Yaskawa INFORM job: R2_W27-A4(90,180)_MP_OK.JBI

/JOB
//NAME R2_W27-A4(90,180)_MP_OK
///FOLDERNAME MP_TEST
//POS
///NPOS 81,81,0,3,0,0
///TOOL 0
///POSTYPE PULSE
///PULSE
C00000=44200,21638,-8218,30156,108783,8626
C00001=67595,-7097,-4564,35957,72928,-14479
C00002=80598,-11631,1969,12944,68774,-20478
C00003=80599,-10712,4409,13031,67770,-20590
C00004=80598,-10715,4407,13031,67770,-20590
C00005=80598,-10719,4404,13032,67770,-20590
C00006=80598,-10715,4407,13031,67770,-20590
C00007=80591,-10742,4386,13033,67770,-20593
C00008=80591,-10741,4387,13033,67770,-20593
C00009=80591,-10742,4386,13033,67770,-20593
C00010=80616,-10653,4455,1959,54638,1214
C00011=74713,-5814,6866,11718,60472,-1274
C00012=77733,-8416,5583,7275,56956,-133
C00013=74892,-4761,7835,12151,60366,-1228
C00014=80616,-10653,4455,1959,54638,1214
C00015=80621,-10639,4466,1958,54638,1216
C00016=80622,-10633,4471,1957,54639,1217
C00017=80626,-10617,4483,1955,54639,1218
C00018=80604,-16221,-12250,12512,75016,-19809
C00019=80613,-16483,-13492,4814,52988,-77020
C00020=80617,-10651,4457,5429,44969,-77444
C00021=80614,-10662,4448,5430,44969,-77445
C00022=79334,-14584,3986,9291,39946,-78705
C00023=81168,-10487,5664,5147,44277,-77224
C00024=80549,-11563,2448,5400,45738,-77430
C00025=81469,-7152,9286,7523,40651,-76865
C00026=81214,-8593,7267,7629,41172,-76947
C00027=79900,-12351,2214,8365,42469,-77481
C00028=78759,-13697,-9805,5892,52278,-77840
C00029=77858,-26804,-24776,6192,54811,-78068
C00030=77858,-26804,-24776,6192,54811,8206
C00031=80560,-10852,4301,23089,88681,-39643
C00032=80562,-10848,4304,23089,88680,-39643
C00033=80600,-11026,3471,23097,89058,-39557
C00034=80047,-12757,2574,23029,88900,-39787
C00035=79798,-9411,5485,22999,88903,-39877
C00036=73696,-20114,6682,31978,77502,-45766
C00037=72021,-21514,1829,31651,80058,-45695
C00038=88031,-24585,-19769,24865,79157,-46389
C00039=74088,-80099,-54440,46439,68409,-50026
C00040=71054,-82284,-78741,37326,78086,-53143
C00041=71054,-82284,-78741,37326,78086,-53143
C00042=141655,19461,21674,-54626,60929,-83209
C00043=140768,21158,24027,-54713,60067,-83168
C00044=140773,21783,25908,-55104,59574,-82809
C00045=140768,21158,24027,-54713,60067,-83168
C00046=156074,19906,-10403,-52836,81444,-87755
C00047=155321,18966,-11276,-52620,81066,-87928
C00048=156074,19906,-10403,-52836,81444,-87755
C00049=158287,-4573,8654,-106143,62454,-35624
C00050=145346,15241,-15914,-44032,85995,9611
C00051=145082,17275,-14042,-43967,85792,9582
C00052=145346,15241,-15914,-44032,85995,9611
C00053=128597,-2596,-22816,-39758,74552,6944
C00054=106236,1119,-8655,-33108,59628,2381
C00055=100502,1007,-8349,-30553,57262,531
C00056=121335,-11193,4016,-73235,33107,-65970
C00057=121314,-11175,4070,-52209,41640,-77705
C00058=121322,-11192,4065,-52217,41640,-77699
C00059=121326,-11199,4064,-52221,41641,-77697
C00060=121319,-11903,2209,-51536,42130,-78112
C00061=122361,-11180,4070,-52628,42228,-77380
C00062=121327,-11199,4064,-52222,41641,-77696
C00063=121327,-11199,4064,-52222,41641,-77696
C00064=121328,-11199,4065,-52223,41641,-77696
C00065=121325,-11192,4067,-52219,41641,-77698
C00066=121317,-11174,4072,-52211,41640,-77704
C00067=121324,-11180,4031,-66023,34984,-69858
C00068=121305,-11164,4064,-33775,34107,58027
C00069=121211,-10931,3851,-41868,44478,53115
C00070=117301,-6994,3549,-31202,46743,49457
C00071=117109,-6013,5862,-33344,45913,49803
C00072=121892,-11860,2463,-42413,44821,53021
C00073=122357,-11331,3957,-43061,44562,53464
C00074=117366,750,11411,-33444,46067,49884
C00075=119475,-2324,8124,-34252,47278,50538
C00076=123076,-13488,2301,-43433,44847,53751
C00077=121299,-11171,4074,-39219,33281,58177
C00078=129161,-93141,-40285,-63646,27916,71647
C00079=59909,-160831,-87956,-63646,27916,71647
C00080=39710,-191418,-114720,-5142,50077,71647
BC00000=114828,232249,1075169
BC00001=111963,174209,1075173
BC00002=110304,140592,1075175
BC00003=109200,135830,1065059
BC00004=108759,133925,1056755
BC00005=108743,133924,1048690
BC00006=108759,133925,1056755
BC00007=119290,133339,1053953
BC00008=118788,131086,1053965
BC00009=119290,133339,1053953
BC00010=81395,143067,1043817
BC00011=79666,135317,1043859
BC00012=81999,134825,1043807
BC00013=81144,135003,1043826
BC00014=81395,143067,1043817
BC00015=73310,143561,1032388
BC00016=72136,145534,1039614
BC00017=69199,150466,1057682
BC00018=110304,140592,1075175
BC00019=82308,150049,1075175
BC00020=81837,149958,1052280
BC00021=81780,147780,1026500
BC00022=81757,146909,1016188
BC00023=81757,146909,1016188
BC00024=81757,146909,1016188
BC00025=81757,146909,1016188
BC00026=81757,146909,1016188
BC00027=81757,146909,1016188
BC00028=82300,142177,1075175
BC00029=82308,150049,1075175
BC00030=82308,150049,1075175
BC00031=162842,108215,1047947
BC00032=157631,106152,1028943
BC00033=155546,105326,1021342
BC00034=155546,105326,1021342
BC00035=155546,105326,1021342
BC00036=155546,105326,1021342
BC00037=155546,105326,1021342
BC00038=169608,133925,979206
BC00039=162842,108215,1047947
BC00040=169608,248553,979206
BC00041=169608,248553,42321
BC00042=261853,172349,216144
BC00043=261853,172349,216144
BC00044=261853,172349,216144
BC00045=261853,172349,216144
BC00046=307725,162058,22582
BC00047=307725,162058,22582
BC00048=307725,162058,22582
BC00049=299050,167122,35683
BC00050=289567,172657,50003
BC00051=289567,172657,50003
BC00052=289567,172657,50003
BC00053=232126,164256,101248
BC00054=174559,155898,152583
BC00055=158444,154728,159769
BC00056=191752,205444,198110
BC00057=212977,154819,280459
BC00058=218243,152180,262530
BC00059=220349,151125,255359
BC00060=220349,151125,255359
BC00061=220349,151125,255359
BC00062=220340,146516,255365
BC00063=220339,146083,255365
BC00064=220329,141475,255371
BC00065=218223,142530,262543
BC00066=212957,145169,280472
BC00067=194357,200564,228108
BC00068=206310,183138,286705
BC00069=214934,140825,283714
BC00070=214934,140825,283714
BC00071=214934,140825,283714
BC00072=221705,136683,270833
BC00073=221705,136683,270833
BC00074=214934,140825,283714
BC00075=214934,140825,283714
BC00076=212593,134321,287024
BC00077=215962,184468,300457
BC00078=215962,184468,300457
BC00079=215962,184468,300457
BC00080=225321,288951,754221
///POSTYPE BASE
///RECTAN
///RCONF 0,0,0,0,0,0,0,0,0,0,0,0,0,0,0,0,0,0,0,0,0,0,0,0
P00001=2714.263,6838.284,-998.276,27.8833,45.1566,-82.5967
P00006=0.222,-3.123,-1.508,0.0000,0.0000,0.0000
P00014=-0.708,0.505,-8.393,0.0000,0.0000,0.0000
//INST
///DATE 2023/11/16 10:53
///ATTR SC,RW
///GROUP1 RB1,BS1
NOP
'r2_W27-A4(90,180)
'
'Path S896
SFTOF
MOVJ C00000 BC00000 VJ=20.00
MOVJ C00001 BC00001 VJ=20.00
MOVL C00002 BC00002 V=100.0
MOVL C00003 BC00003 V=100.0
MOVL C00004 BC00004 V=60.0
REFP 3 C00005 BC00005
CALL JOB:SEARCH-R1
SET P014 P006
SFTON P014
MOVL C00006 BC00006 V=60.0
MOVL C00007 BC00007 V=60.0
REFP 3 C00008 BC00008
CALL JOB:SEARCH-R1
SET P014 P006
SFTON P014
MOVL C00009 BC00009 V=60.0
MOVL C00010 BC00010 V=100.0
MOVL C00011 BC00011 V=60.0
REFP 3 C00012 BC00012
CALL JOB:SEARCH-R1
SET P014 P006
SFTON P014
MOVL C00013 BC00013 V=60.0
MOVL C00014 BC00014 V=100.0
MOVL C00015 BC00015 V=100.0
MOVL C00016 BC00016 V=100.0
MOVL C00017 BC00017 V=100.0
'Path VIA902
SFTOF
MOVJ C00018 BC00018 VJ=20.00
'Path W898
SFTOF
SFTON P014
MOVJ C00019 BC00019 VJ=20.00
MOVJ C00020 BC00020 VJ=20.00
MOVL C00021 BC00021 V=100.0
MOVL C00022 BC00022 V=100.0 PL=0
REFP 1 C00023 BC00023
REFP 2 C00024 BC00024
MACRO1 MJ#(0) ARGF7
ARCON
MOVL C00025 BC00025 V=10.8
ARCOF
MOVL C00026 BC00026 V=100.0
MOVL C00027 BC00027 V=100.0
MOVL C00028 BC00028 V=100.0
SFTOF
'Path VIA903
SFTOF
MOVJ C00029 BC00029 VJ=20.00
'Path VIA904
SFTOF
MOVJ C00030 BC00030 VJ=20.00
'Path W901
SFTOF
SFTON P014
MOVJ C00031 BC00031 VJ=20.00
MOVL C00032 BC00032 V=100.0
MOVL C00033 BC00033 V=100.0 PL=0
REFP 1 C00034 BC00034
REFP 2 C00035 BC00035
MACRO1 MJ#(0) ARGF6
ARCON
MOVL C00036 BC00036 V=12.5
ARCOF
MOVL C00037 BC00037 V=100.0
MOVL C00038 BC00038 V=100.0
SFTOF
'Path VIA907
SFTOF
MOVJ C00039 BC00039 VJ=20.00
'Path VIA905
SFTOF
MOVJ C00040 BC00040 VJ=20.00
CALL JOB:CLEAN-R1_LONG
'Path VIA906
SFTOF
MOVJ C00041 BC00041 VJ=20.00
'Path S845
SFTOF
MOVL C00042 BC00042 V=100.0
MOVL C00043 BC00043 V=60.0
REFP 3 C00044 BC00044
CALL JOB:SEARCH-R1
SET P001 P006
SFTON P001
MOVL C00045 BC00045 V=60.0
MOVL C00046 BC00046 V=60.0
REFP 3 C00047 BC00047
CALL JOB:SEARCH-R1
SET P001 P006
SFTON P001
MOVL C00048 BC00048 V=60.0
MOVL C00049 BC00049 V=100.0
MOVL C00050 BC00050 V=60.0
REFP 3 C00051 BC00051
CALL JOB:SEARCH-R1
SET P001 P006
SFTON P001
MOVL C00052 BC00052 V=60.0
MOVL C00053 BC00053 V=100.0
MOVL C00054 BC00054 V=100.0
MOVL C00055 BC00055 V=100.0
'Path W846
SFTOF
SFTON P001
MOVJ C00056 BC00056 VJ=20.00
MOVL C00057 BC00057 V=100.0
MOVL C00058 BC00058 V=100.0
MOVL C00059 BC00059 V=100.0 PL=0
REFP 1 C00060 BC00060
REFP 2 C00061 BC00061
MACRO1 MJ#(0) ARGF0
COMM ARCON
MOVL C00062 BC00062 V=10.0
MOVL C00063 BC00063 V=10.0
MOVL C00064 BC00064 V=10.0
ARCOF
MOVL C00065 BC00065 V=100.0
MOVL C00066 BC00066 V=100.0
MOVL C00067 BC00067 V=100.0
SFTOF
'Path W847
SFTOF
SFTON P001
MOVJ C00068 BC00068 VJ=20.00
MOVL C00069 BC00069 V=100.0
MOVL C00070 BC00070 V=100.0
MOVL C00071 BC00071 V=100.0 PL=0
REFP 1 C00072 BC00072
REFP 2 C00073 BC00073
MACRO1 MJ#(0) ARGF7
ARCON
MOVL C00074 BC00074 V=10.8
ARCOF
MOVL C00075 BC00075 V=100.0
MOVL C00076 BC00076 V=100.0
MOVL C00077 BC00077 V=100.0
SFTOF
MOVJ C00078 BC00078 VJ=20.00
MOVJ C00079 BC00079 VJ=20.00
MOVJ C00080 BC00080 VJ=20.00
END
